// TIA Portal project "CONTROL_ENERGIA" (V12)

(* hardware
DEVICE "S7-300 station_2"  S7-300 station
   slot 0: "Perfil soporte_0"  Rail  6ES7 390-1***0-0AA0
   slot 1: "PS 307 5A_1"  PS 307 5A  6ES7 307-1EA00-0AA0
   slot 2: "CONTROL_ENERGIA"  CPU 314C-2 PN/DP  6ES7 314-6EH04-0AB0  V3.3
      slot 2: "Interfaz PROFINET_1"  PN-IO
         slot 1: "Port_1"  Port
         slot 2: "Port_2"  Port
      slot 5: "DI24/DO16_1"  DI24/DO16
      slot 6: "AI5/AO2_1"  AI5/AO2
      slot 7: "Contaje_1"  Counter
      slot 8: "Posicionamiento_1"  Positioning
   slot 4: "DI8/DO8 x 24V DC / 0,5A_1"  DI8/DO8xDC24V/0.5A  6ES7 323-1BH01-0AA0
*)

// ===== PLC "CONTROL_ENERGIA"  CPU 314C-2 PN/DP =====

VAR_GLOBAL   // PLC tag table "Tabla de variables estándar"
   "Tag_1" AT %I136.0 : Bool;
   "Tag_2" AT %Q136.0 : Bool;
   "Tag_3" AT %I137.0 : Bool;
   "Tag_4" AT %Q136.1 : Bool;
   "Tag_5" AT %I138.0 : Bool;
   "Tag_6" AT %Q137.2 : Bool;
   "Tag_7" AT %Q136.2 : Bool;
   "Tag_8" AT %Q137.0 : Bool;
   "shunt_corriente" AT %IW800 : Int;
   "Tag_10" AT %MW10 : Word;
   "intensidad_medida" AT %MD12 : Real;
   "siempre_cero" AT %M254.0 : Bool;
   "Tag_13" AT %QW800 : Int;
   "Tag_14" AT %MD55 : DWord;
   "consigna salida" AT %MW60 : Int;
   "error_2" AT %MW62 : Word;
   "siempre_uno" AT %M254.1 : Bool;
   "x" AT %MD10 : Real;
   "y" AT %MD20 : Real;
   "x_ala_y" AT %MD30 : Real;
   "intensidad" AT %MD40 : Real;
   "horas" AT %MD50 : Real;
   "intensidad_compensada_peukert" AT %MD60 : Real;
   "rendimiento" AT %MD70 : Real;
   "recarga" AT %MD80 : Real;
   "ret_val_unscale" AT %MW100 : Word;
   "SOC" AT %MD90 : Real;
END_VAR

DATA_BLOCK "parametros_configuracion"   // DB1
{ S7_Optimized_Access := 'FALSE' }
VERSION : 0.1
   VAR
      marca_encendido : Bool;
      Capacidad_fabricante : Real := 625.0;
      Tasa_segun_fabricante : Real := 10.0;
      coeficiente_peukert : Real := 1.13;
      rendimiento_carga : Real := 90.0;
   END_VAR
BEGIN
END_DATA_BLOCK

DATA_BLOCK "Calculo_capacidad_peukert_DB"   // DB2
{ S7_Optimized_Access := 'FALSE' }
VERSION : 0.1
// stored: InstanceOfName Calculo_capacidad_peukert
"Calculo_capacidad_peukert"
BEGIN
END_DATA_BLOCK

DATA_BLOCK "x_a_la_y_DB_intensidad"   // DB3
{ S7_Optimized_Access := 'FALSE' }
VERSION : 0.1
// stored: InstanceOfName x_a_la_y
"x_a_la_y"
BEGIN
END_DATA_BLOCK

DATA_BLOCK "x_a_la_y_DB_capacidad"   // DB4
{ S7_Optimized_Access := 'FALSE' }
VERSION : 0.1
// stored: InstanceOfName x_a_la_y
"x_a_la_y"
BEGIN
END_DATA_BLOCK

DATA_BLOCK "Intensidad_compensada_peukert_DB"   // DB5
{ S7_Optimized_Access := 'FALSE' }
VERSION : 0.1
// stored: InstanceOfName Intensidad_consumida_compensada_peukert
"Intensidad_consumida_compensada_peukert"
BEGIN
END_DATA_BLOCK

DATA_BLOCK "Intensidad_recargada_DB"   // DB6
{ S7_Optimized_Access := 'FALSE' }
VERSION : 0.1
// stored: InstanceOfName Intensidad_recargada
"Intensidad_recargada"
BEGIN
END_DATA_BLOCK

DATA_BLOCK "balance_energetico_DB"   // DB7
{ S7_Optimized_Access := 'FALSE' }
VERSION : 0.1
// stored: InstanceOfName balance_energetico
"balance_energetico"
BEGIN
END_DATA_BLOCK

DATA_BLOCK "S.O.C_DB"   // DB8
{ S7_Optimized_Access := 'FALSE' }
VERSION : 0.1
// stored: InstanceOfName S.O.C
"S.O.C"
BEGIN
END_DATA_BLOCK

FUNCTION_BLOCK "Calculo_capacidad_peukert"   // FB1, LAD
TITLE = calcula por fases la capacidad estandarizada segun peukert Cp=R(C/R)^n
{ S7_Optimized_Access := 'FALSE' }
VERSION : 0.1
   VAR_INPUT
      C : Real;
      R : Real;
      n : Real;
   END_VAR
   VAR_OUTPUT
      CP : Real;
   END_VAR
   VAR_IN_OUT
      "cociente_C/R" : Real;
      parentesis : Real;
   END_VAR
BEGIN

REGION Network 1: Calcula el cociente C/R
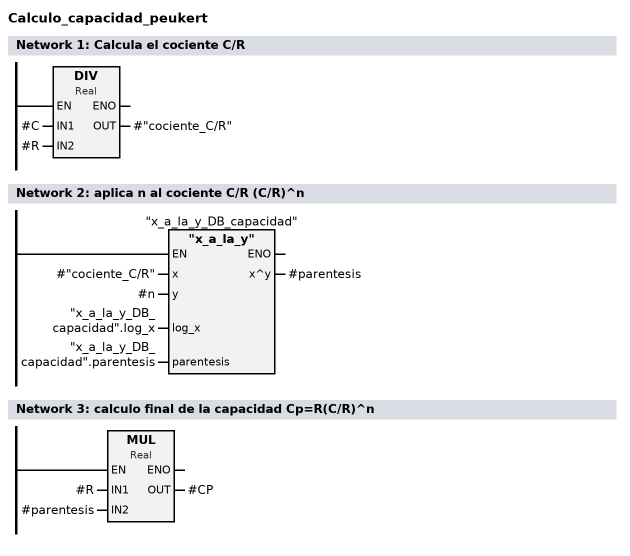
   RUNG wire#powerrail
      { S7_Templates := "SrcType := Real"; S7_GenerateENO := "TRUE" } Div(in1 := #C, in2 := #R, out => #"cociente_C/R")
   END_RUNG
   // the same network as SCL:
   #"cociente_C/R" := #C / #R;
END_REGION

REGION Network 2: aplica n al cociente C/R (C/R)^n
   RUNG wire#powerrail
      "x_a_la_y_DB_capacidad"(x := #"cociente_C/R", y := #n, log_x := "x_a_la_y_DB_capacidad".log_x, parentesis := "x_a_la_y_DB_capacidad".parentesis, "x^y" => #parentesis)
   END_RUNG
   // the same network as SCL:
   "x_a_la_y_DB_capacidad"(x := #"cociente_C/R",   // "x_a_la_y"
                           y := #n,
                           log_x := "x_a_la_y_DB_capacidad".log_x,
                           parentesis := "x_a_la_y_DB_capacidad".parentesis,
                           "x^y" => #parentesis);
END_REGION

REGION Network 3: calculo final de la capacidad Cp=R(C/R)^n
   RUNG wire#powerrail
      { S7_Templates := "SrcType := Real"; S7_GenerateENO := "TRUE" } Mul(in1 := #R, in2 := #parentesis, out => #CP)
   END_RUNG
   // the same network as SCL:
   #CP := #R * #parentesis;
END_REGION
END_FUNCTION_BLOCK

FUNCTION_BLOCK "lectura_intensidad_real"   // FB2, LAD
TITLE = lectura de la intensidad sin compensar
{ S7_Optimized_Access := 'FALSE' }
VERSION : 0.1
BEGIN

REGION Network 1: lectura de la intensidad
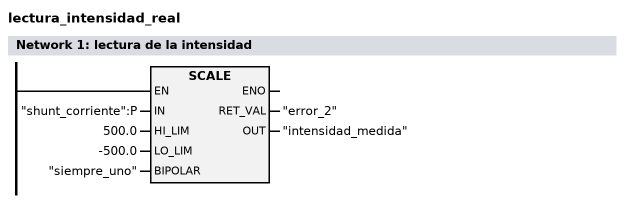
   "error_2" := SCALE(IN := "shunt_corriente":P,
                      HI_LIM := 500.0,
                      LO_LIM := -500.0,
                      BIPOLAR := "siempre_uno",
                      OUT => "intensidad_medida");
END_REGION
END_FUNCTION_BLOCK

FUNCTION_BLOCK "x_a_la_y"   // FB3, LAD
TITLE = calcular trampeando X^Y=EXP(Y*LOG(X))
{ S7_Optimized_Access := 'FALSE' }
VERSION : 0.1
   VAR_INPUT
      x : Real;
      y : Real;
   END_VAR
   VAR_OUTPUT
      "x^y" : Real;
   END_VAR
   VAR_IN_OUT
      log_x : Real;
      parentesis : Real;
   END_VAR
BEGIN

REGION Network 1: LOG(X)
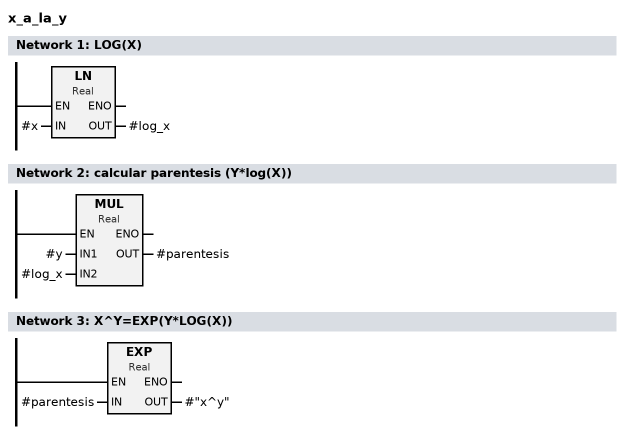
   #log_x := LN(#x);
END_REGION

REGION Network 2: calcular parentesis (Y*log(X))
   RUNG wire#powerrail
      { S7_Templates := "SrcType := Real"; S7_GenerateENO := "TRUE" } Mul(in1 := #y, in2 := #log_x, out => #parentesis)
   END_RUNG
   // the same network as SCL:
   #parentesis := #y * #log_x;
END_REGION

REGION Network 3: X^Y=EXP(Y*LOG(X))
   #"x^y" := EXP(#parentesis);
END_REGION
END_FUNCTION_BLOCK

FUNCTION_BLOCK "Intensidad_consumida_compensada_peukert"   // FB4, LAD
TITLE = Capacidad consumida compensada por Peukert Cp=T*I^n
{ S7_Optimized_Access := 'FALSE' }
VERSION : 0.1
   VAR_INPUT
      tiempo_consumo_horas : Real;
      n : Real;
      intensidad_consumida_amperios : Real;
   END_VAR
   VAR_OUTPUT
      intensidad_compensada : Real;
   END_VAR
   VAR_IN_OUT
      potencia : Real;
      intensidad_absoluta : Real;
   END_VAR
BEGIN

REGION Network 1: sacar el valor absoluto de la I Valores negativos conducen a error
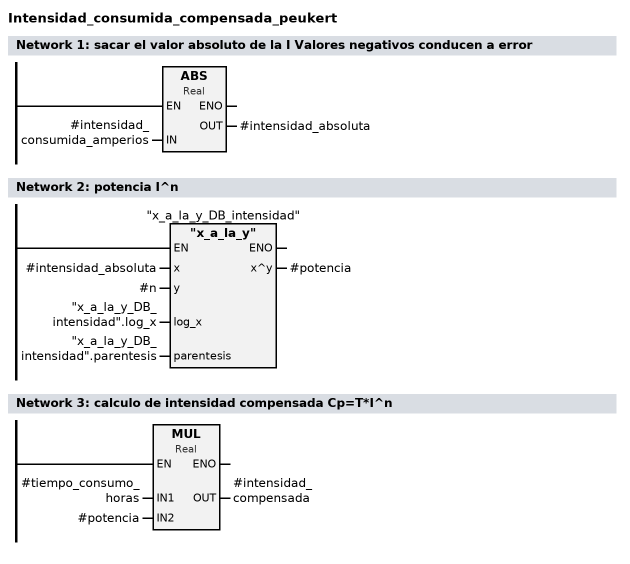
   RUNG wire#powerrail
      { S7_Templates := "SrcType := Real"; S7_GenerateENO := "TRUE" } Abs(in := #intensidad_consumida_amperios, out => #intensidad_absoluta)
   END_RUNG
   // the same network as SCL:
   #intensidad_absoluta := ABS(#intensidad_consumida_amperios);
END_REGION

REGION Network 2: potencia I^n
   RUNG wire#powerrail
      "x_a_la_y_DB_intensidad"(x := #intensidad_absoluta, y := #n, log_x := "x_a_la_y_DB_intensidad".log_x, parentesis := "x_a_la_y_DB_intensidad".parentesis, "x^y" => #potencia)
   END_RUNG
   // the same network as SCL:
   "x_a_la_y_DB_intensidad"(x := #intensidad_absoluta,   // "x_a_la_y"
                           y := #n,
                           log_x := "x_a_la_y_DB_intensidad".log_x,
                           parentesis := "x_a_la_y_DB_intensidad".parentesis,
                           "x^y" => #potencia);
END_REGION

REGION Network 3: calculo de intensidad compensada Cp=T*I^n
   RUNG wire#powerrail
      { S7_Templates := "SrcType := Real"; S7_GenerateENO := "TRUE" } Mul(in1 := #tiempo_consumo_horas, in2 := #potencia, out => #intensidad_compensada)
   END_RUNG
   // the same network as SCL:
   #intensidad_compensada := #tiempo_consumo_horas * #potencia;
END_REGION
END_FUNCTION_BLOCK

FUNCTION_BLOCK "Intensidad_recargada"   // FB5, LAD
TITLE = intensidad entrante aplicado el rendimiento recarga = I*0,X%*tiempo_transcurrido
{ S7_Optimized_Access := 'FALSE' }
VERSION : 0.1
   VAR_INPUT
      intensidad : Real;
      rendimiento : Real;
      tiempo : Real;
   END_VAR
   VAR_IN_OUT
      recarga : Real;
   END_VAR
BEGIN

REGION Network 1: aplica a la recarga el rendimiento configurado
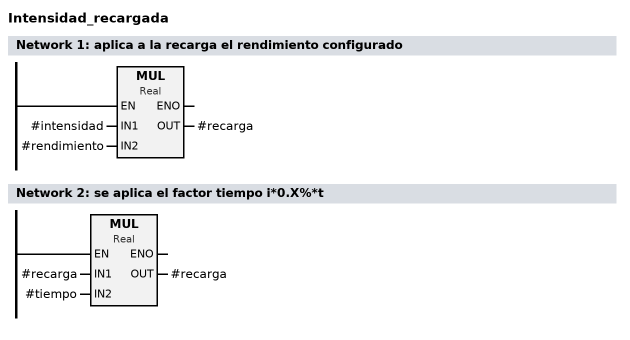
   RUNG wire#powerrail
      { S7_Templates := "SrcType := Real"; S7_GenerateENO := "TRUE" } Mul(in1 := #intensidad, in2 := #rendimiento, out => #recarga)
   END_RUNG
   // the same network as SCL:
   #recarga := #intensidad * #rendimiento;
END_REGION

REGION Network 2: se aplica el factor tiempo i*0.X%*t
   RUNG wire#powerrail
      { S7_Templates := "SrcType := Real"; S7_GenerateENO := "TRUE" } Mul(in1 := #recarga, in2 := #tiempo, out => #recarga)
   END_RUNG
   // the same network as SCL:
   #recarga := #recarga * #tiempo;
END_REGION
END_FUNCTION_BLOCK

FUNCTION_BLOCK "balance_energetico"   // FB6, LAD
TITLE = calcula el balance energetico segun peukert y rendimiento ajustados en parametros
{ S7_Optimized_Access := 'FALSE' }
VERSION : 0.1
   VAR_INPUT
      intensidad_real : Real;
      intensidad_peukert : Real;
      intensidad_carga_comp : Real;
   END_VAR
   VAR_IN_OUT
      intensidad_acumulada : Real;
   END_VAR
BEGIN

REGION Network 1: incrementa la Int acumulada con la int cargada compensada con el rendimiento
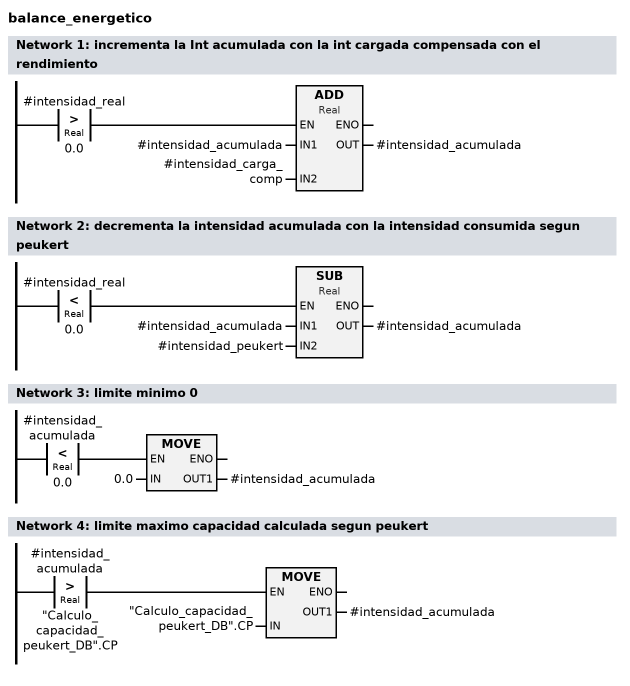
   RUNG wire#powerrail
      { S7_Templates := "SrcType := Real" } GT_Contact(in1 := #intensidad_real, in2 := 0.0)
      { S7_Templates := "SrcType := Real"; S7_GenerateENO := "TRUE" } Add(in1 := #intensidad_acumulada, in2 := #intensidad_carga_comp, out => #intensidad_acumulada)
   END_RUNG
   // the same network as SCL:
   IF #intensidad_real > 0.0 THEN
       #intensidad_acumulada := #intensidad_acumulada + #intensidad_carga_comp;
   END_IF;
END_REGION

REGION Network 2: decrementa la intensidad acumulada con la intensidad consumida segun peukert
   RUNG wire#powerrail
      { S7_Templates := "SrcType := Real" } LT_Contact(in1 := #intensidad_real, in2 := 0.0)
      { S7_Templates := "SrcType := Real"; S7_GenerateENO := "TRUE" } Sub(in1 := #intensidad_acumulada, in2 := #intensidad_peukert, out => #intensidad_acumulada)
   END_RUNG
   // the same network as SCL:
   IF #intensidad_real < 0.0 THEN
       #intensidad_acumulada := #intensidad_acumulada - #intensidad_peukert;
   END_IF;
END_REGION

REGION Network 3: limite minimo 0
   RUNG wire#powerrail
      { S7_Templates := "SrcType := Real" } LT_Contact(in1 := #intensidad_acumulada, in2 := 0.0)
      { S7_GenerateENO := "TRUE" } Move(in := 0.0, out1 => #intensidad_acumulada)
   END_RUNG
   // the same network as SCL:
   IF #intensidad_acumulada < 0.0 THEN #intensidad_acumulada := 0.0; END_IF;
END_REGION

REGION Network 4: limite maximo capacidad calculada segun peukert
   RUNG wire#powerrail
      { S7_Templates := "SrcType := Real" } GT_Contact(in1 := #intensidad_acumulada, in2 := "Calculo_capacidad_peukert_DB".CP)
      { S7_GenerateENO := "TRUE" } Move(in := "Calculo_capacidad_peukert_DB".CP, out1 => #intensidad_acumulada)
   END_RUNG
   // the same network as SCL:
   IF #intensidad_acumulada > "Calculo_capacidad_peukert_DB".CP THEN
       #intensidad_acumulada := "Calculo_capacidad_peukert_DB".CP;
   END_IF;
END_REGION
END_FUNCTION_BLOCK

FUNCTION_BLOCK "S.O.C"   // FB7, LAD
{ S7_Optimized_Access := 'FALSE' }
VERSION : 0.1
   VAR_INPUT
      "intensidad_acumulada." : Real;
   END_VAR
   VAR_OUTPUT
      SOC : Real;
   END_VAR
   VAR_IN_OUT
      intensidad_integer : Int;
   END_VAR
BEGIN

REGION Network 1: convertimos la intensidad de real a entero
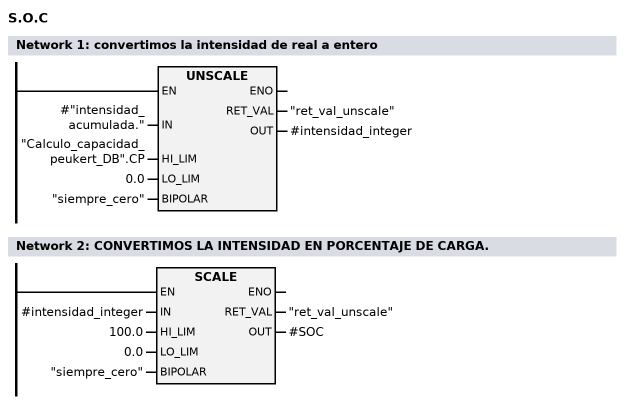
   "ret_val_unscale" := UNSCALE(IN := #"intensidad_acumulada.",
                           HI_LIM := "Calculo_capacidad_peukert_DB".CP,
                           LO_LIM := 0.0,
                           BIPOLAR := "siempre_cero",
                           OUT => #intensidad_integer);
END_REGION

REGION Network 2: CONVERTIMOS LA INTENSIDAD EN PORCENTAJE DE CARGA.
   "ret_val_unscale" := SCALE(IN := #intensidad_integer,
                           HI_LIM := 100.0,
                           LO_LIM := 0.0,
                           BIPOLAR := "siempre_cero",
                           OUT => #SOC);
END_REGION
END_FUNCTION_BLOCK

ORGANIZATION_BLOCK "Main"   // OB1, LAD
TITLE = "Main Program Sweep (Cycle)"
{ S7_Optimized_Access := 'FALSE' }
VERSION : 0.1
   VAR_TEMP
      OB1_EV_CLASS : Byte;   // Bits 0-3 = 1 (Coming event), Bits 4-7 = 1 (Event class 1)
      OB1_SCAN_1 : Byte;   // 1 (Cold restart scan 1 of OB 1), 3 (Scan 2-n of OB 1)
      OB1_PRIORITY : Byte;   // Priority of OB Execution
      OB1_OB_NUMBR : Byte;   // 1 (Organization block 1, OB1)
      OB1_RESERVED_1 : Byte;   // Reserved for system
      OB1_RESERVED_2 : Byte;   // Reserved for system
      OB1_PREV_CYCLE : Int;   // Cycle time of previous OB1 scan (milliseconds)
      OB1_MIN_CYCLE : Int;   // Minimum cycle time of OB1 (milliseconds)
      OB1_MAX_CYCLE : Int;   // Maximum cycle time of OB1 (milliseconds)
      OB1_DATE_TIME : Date_And_Time;   // Date and time OB1 started
   END_VAR
BEGIN

REGION Network 1: prueba calculo capacidad peukert
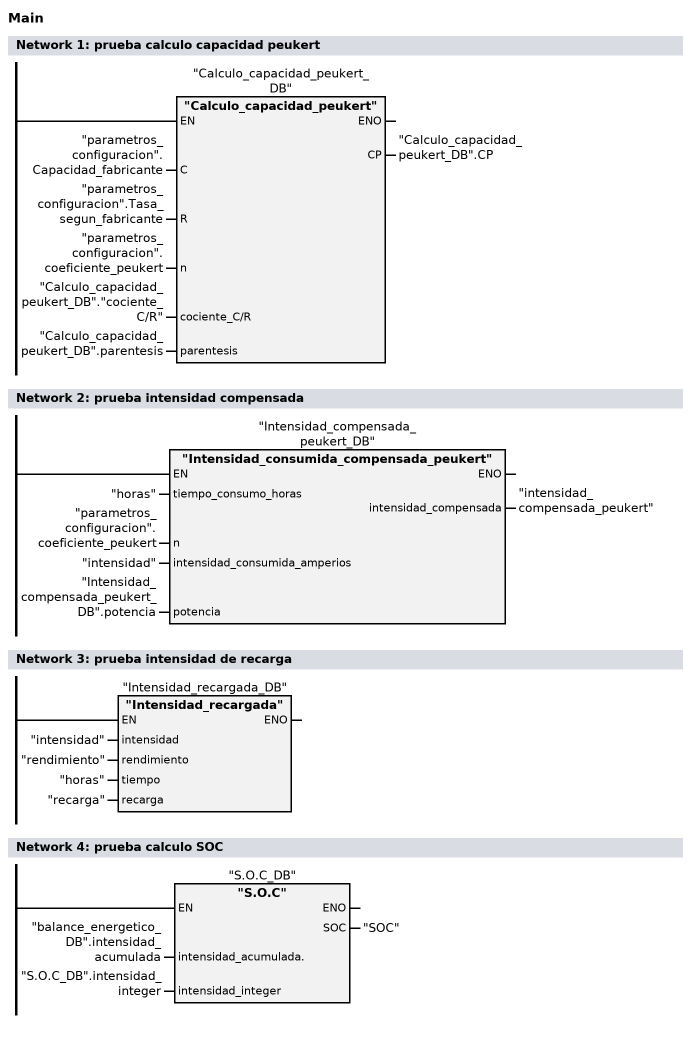
   RUNG wire#powerrail
      "Calculo_capacidad_peukert_DB"(C := "parametros_configuracion".Capacidad_fabricante, R := "parametros_configuracion".Tasa_segun_fabricante, n := "parametros_configuracion".coeficiente_peukert, "cociente_C/R" := "Calculo_capacidad_peukert_DB"."cociente_C/R", parentesis := "Calculo_capacidad_peukert_DB".parentesis, CP => "Calculo_capacidad_peukert_DB".CP)
   END_RUNG
   // the same network as SCL:
   "Calculo_capacidad_peukert_DB"(C := "parametros_configuracion".Capacidad_fabricante,   // "Calculo_capacidad_peukert"
                           R := "parametros_configuracion".Tasa_segun_fabricante,
                           n := "parametros_configuracion".coeficiente_peukert,
                           "cociente_C/R" := "Calculo_capacidad_peukert_DB"."cociente_C/R",
                           parentesis := "Calculo_capacidad_peukert_DB".parentesis,
                           CP => "Calculo_capacidad_peukert_DB".CP);
END_REGION

REGION Network 2: prueba intensidad compensada
   RUNG wire#powerrail
      "Intensidad_compensada_peukert_DB"(tiempo_consumo_horas := "horas", n := "parametros_configuracion".coeficiente_peukert, potencia := "Intensidad_compensada_peukert_DB".potencia, intensidad_consumida_amperios := "intensidad", intensidad_compensada => "intensidad_compensada_peukert")
   END_RUNG
   // the same network as SCL:
   "Intensidad_compensada_peukert_DB"(tiempo_consumo_horas := "horas",   // "Intensidad_consumida_compensada_peukert"
                           n := "parametros_configuracion".coeficiente_peukert,
                           intensidad_consumida_amperios := "intensidad",
                           potencia := "Intensidad_compensada_peukert_DB".potencia,
                           intensidad_compensada => "intensidad_compensada_peukert");
END_REGION

REGION Network 3: prueba intensidad de recarga
   RUNG wire#powerrail
      "Intensidad_recargada_DB"(intensidad := "intensidad", rendimiento := "rendimiento", tiempo := "horas", recarga := "recarga")
   END_RUNG
   // the same network as SCL:
   "Intensidad_recargada_DB"(intensidad := "intensidad",   // "Intensidad_recargada"
                           rendimiento := "rendimiento",
                           tiempo := "horas",
                           recarga := "recarga");
END_REGION

REGION Network 4: prueba calculo SOC
   RUNG wire#powerrail
      "S.O.C_DB"("intensidad_acumulada." := "balance_energetico_DB".intensidad_acumulada, intensidad_integer := "S.O.C_DB".intensidad_integer, SOC => "SOC")
   END_RUNG
   // the same network as SCL:
   "S.O.C_DB"("intensidad_acumulada." := "balance_energetico_DB".intensidad_acumulada,   // "S.O.C"
              intensidad_integer := "S.O.C_DB".intensidad_integer,
              SOC => "SOC");
END_REGION
END_ORGANIZATION_BLOCK

ORGANIZATION_BLOCK "SAMPLER"   // OB32, LAD
TITLE = "Cyclic Interrupt"
{ S7_Optimized_Access := 'FALSE' }
VERSION : 0.1
   VAR_TEMP
      OB32_EV_CLASS : Byte;   // Bits 0-3 = 1 (Coming event), Bits 4-7 = 1 (Event class 1)
      OB32_STRT_INF : Byte;   // 16#33 (OB 32 has started)
      OB32_PRIORITY : Byte;   // Priority of OB Execution
      OB32_OB_NUMBR : Byte;   // 32 (Organization block 32, OB32)
      OB32_RESERVED_1 : Byte;   // Reserved for system
      OB32_RESERVED_2 : Byte;   // Reserved for system
      OB32_PHS_OFFSET : Int;   // Phase offset (integer, milliseconds)
      OB32_RESERVED_3 : Int;   // Reserved for system
      OB32_EXC_FREQ : Int;   // Frequency of execution (msec)
      OB32_DATE_TIME : Date_And_Time;   // Date and time OB32 started
   END_VAR
BEGIN

REGION Network 1: calcula balance energetico usando las I calculadas y el factor tiempo (tiempo sampler)
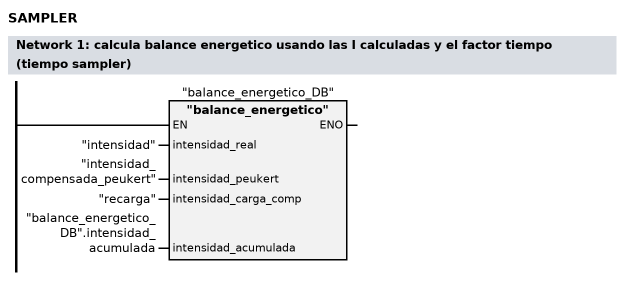
   RUNG wire#powerrail
      "balance_energetico_DB"(intensidad_real := "intensidad", intensidad_peukert := "intensidad_compensada_peukert", intensidad_carga_comp := "recarga", intensidad_acumulada := "balance_energetico_DB".intensidad_acumulada)
   END_RUNG
   // the same network as SCL:
   "balance_energetico_DB"(intensidad_real := "intensidad",   // "balance_energetico"
                           intensidad_peukert := "intensidad_compensada_peukert",
                           intensidad_carga_comp := "recarga",
                           intensidad_acumulada := "balance_energetico_DB".intensidad_acumulada);
END_REGION
END_ORGANIZATION_BLOCK

ORGANIZATION_BLOCK "CYCL_FLT"   // OB80, LAD
TITLE = "Cycle Time Fault"
{ S7_Optimized_Access := 'FALSE' }
VERSION : 0.1
   VAR_TEMP
      OB80_EV_CLASS : Byte;   // 16#35, Event class 3, Entering event state, Internal fault event
      OB80_FLT_ID : Byte;   // 16#XX, Fault identifcation code
      OB80_PRIORITY : Byte;   // Priority of OB Execution
      OB80_OB_NUMBR : Byte;   // 80 (Organization block 80, OB80)
      OB80_RESERVED_1 : Byte;   // Reserved for system
      OB80_RESERVED_2 : Byte;   // Reserved for system
      OB80_ERROR_INFO : Word;   // Error information on event
      OB80_ERR_EV_CLASS : Byte;   // Class of event causing error
      OB80_ERR_EV_NUM : Byte;   // Number of event causing error
      OB80_OB_PRIORITY : Byte;   // Priority of OB causing error
      OB80_OB_NUM : Byte;   // Number of OB causing error
      OB80_DATE_TIME : Date_And_Time;   // Date and time OB80 started
   END_VAR
BEGIN
END_ORGANIZATION_BLOCK

ORGANIZATION_BLOCK "I/O_FLT1"   // OB82, LAD
TITLE = "I/O Point Fault"
{ S7_Optimized_Access := 'FALSE' }
VERSION : 0.1
   VAR_TEMP
      OB82_EV_CLASS : Byte;   // 16#39, Event class 3, Entering event state, Internal fault event
      OB82_FLT_ID : Byte;   // 16#XX, Fault identifcation code
      OB82_PRIORITY : Byte;   // Priority of OB Execution
      OB82_OB_NUMBR : Byte;   // 82 (Organization block 82, OB82)
      OB82_RESERVED_1 : Byte;   // Reserved for system
      OB82_IO_FLAG : Byte;   // Input (01010100), Output (01010101)
      OB82_MDL_ADDR : Word;   // Base address of module with fault
      OB82_MDL_DEFECT : Bool;   // Module defective
      OB82_INT_FAULT : Bool;   // Internal fault
      OB82_EXT_FAULT : Bool;   // External fault
      OB82_PNT_INFO : Bool;   // Point information
      OB82_EXT_VOLTAGE : Bool;   // External voltage low
      OB82_FLD_CONNCTR : Bool;   // Field wiring connector missing
      OB82_NO_CONFIG : Bool;   // Module has no configuration data
      OB82_CONFIG_ERR : Bool;   // Module has configuration error
      OB82_MDL_TYPE : Byte;   // Type of module
      OB82_SUB_MDL_ERR : Bool;   // Sub-Module is missing or has error
      OB82_COMM_FAULT : Bool;   // Communication fault
      OB82_MDL_STOP : Bool;   // Module is stopped
      OB82_WTCH_DOG_FLT : Bool;   // Watch dog timer stopped module
      OB82_INT_PS_FLT : Bool;   // Internal power supply fault
      OB82_PRIM_BATT_FLT : Bool;   // Primary battery is in fault
      OB82_BCKUP_BATT_FLT : Bool;   // Backup battery is in fault
      OB82_RESERVED_2 : Bool;   // Reserved for system
      OB82_RACK_FLT : Bool;   // Rack fault, only for bus interface module
      OB82_PROC_FLT : Bool;   // Processor fault
      OB82_EPROM_FLT : Bool;   // EPROM fault
      OB82_RAM_FLT : Bool;   // RAM fault
      OB82_ADU_FLT : Bool;   // ADU fault
      OB82_FUSE_FLT : Bool;   // Fuse fault
      OB82_HW_INTR_FLT : Bool;   // Hardware interupt input in fault
      OB82_RESERVED_3 : Bool;   // Reserved for system
      OB82_DATE_TIME : Date_And_Time;   // Date and time OB82 started
   END_VAR
BEGIN
END_ORGANIZATION_BLOCK

ORGANIZATION_BLOCK "I/O_FLT2"   // OB83, LAD
TITLE = "I/O Point Fault"
{ S7_Optimized_Access := 'FALSE' }
VERSION : 0.1
   VAR_TEMP
      OB83_EV_CLASS : Byte;   // 16#38/39, Event class 3, module inserted/removed (8/9)
      OB83_FLT_ID : Byte;   // 16#XX, Fault identifcation code
      OB83_PRIORITY : Byte;   // Priority of OB Execution
      OB83_OB_NUMBR : Byte;   // 83 (Organization block 83, OB83)
      OB83_RESERVED_1 : Byte;   // Reserved for system
      OB83_MDL_ID : Byte;   // Input module (01010100), Output module (01010101)
      OB83_MDL_ADDR : Word;   // Base address of module with point fault
      OB83_RACK_NUM : Int;   // Number of rack that has module with point fault
      OB83_MDL_TYPE : Word;   // Module type with point fault
      OB83_DATE_TIME : Date_And_Time;   // Date and time OB83 started
   END_VAR
BEGIN
END_ORGANIZATION_BLOCK

ORGANIZATION_BLOCK "OBNL_FLT"   // OB85, LAD
TITLE = "Organization Block (OB) Not Loaded Fault"
{ S7_Optimized_Access := 'FALSE' }
VERSION : 0.1
   VAR_TEMP
      OB85_EV_CLASS : Byte;   // 16#35 Event class 3
      OB85_FLT_ID : Byte;   // 16#XX, Fault identification code
      OB85_PRIORITY : Byte;   // Priority of OB Execution
      OB85_OB_NUMBR : Byte;   // 85 (Organization block 85, OB85)
      OB85_RESERVED_1 : Byte;   // Reserved for system
      OB85_RESERVED_2 : Byte;   // Reserved for system
      OB85_RESERVED_3 : Int;   // Reserved for system
      OB85_ERR_EV_CLASS : Byte;   // Class of event causing error
      OB85_ERR_EV_NUM : Byte;   // Number of event causing error
      OB85_OB_PRIOR : Byte;   // Priority of OB causing error
      OB85_OB_NUM : Byte;   // Number of OB causing error
      OB85_DATE_TIME : Date_And_Time;   // Date and time OB85 started
   END_VAR
BEGIN
END_ORGANIZATION_BLOCK

ORGANIZATION_BLOCK "COMPLETE RESTART"   // OB100, LAD
TITLE = "Complete Restart"
{ S7_Optimized_Access := 'FALSE' }
VERSION : 0.1
   VAR_TEMP
      OB100_EV_CLASS : Byte;   // 16#13, Event class 1, Entering event state, Event logged in diagnostic buffer
      OB100_STRTUP : Byte;   // 16#81/82/83/84 Method of startup
      OB100_PRIORITY : Byte;   // Priority of OB Execution
      OB100_OB_NUMBR : Byte;   // 100 (Organization block 100, OB100)
      OB100_RESERVED_1 : Byte;   // Reserved for system
      OB100_RESERVED_2 : Byte;   // Reserved for system
      OB100_STOP : Word;   // Event that caused CPU to stop (16#4xxx)
      OB100_STRT_INFO : DWord;   // Information on how system started
      OB100_DATE_TIME : Date_And_Time;   // Date and time OB100 started
   END_VAR
BEGIN

REGION Network 1: Crear Cero
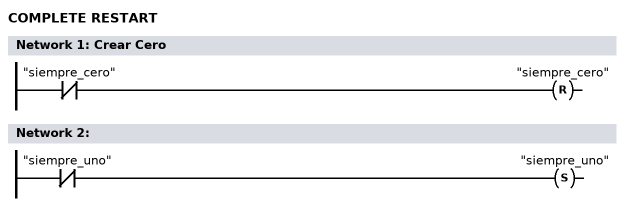
   RUNG wire#powerrail
      I_Contact( "siempre_cero" )
      R_Coil( "siempre_cero" )
   END_RUNG
   // the same network as SCL:
   IF NOT "siempre_cero" THEN "siempre_cero" := FALSE; END_IF;
END_REGION

REGION Network 2
   RUNG wire#powerrail
      I_Contact( "siempre_uno" )
      S_Coil( "siempre_uno" )
   END_RUNG
   // the same network as SCL:
   IF NOT "siempre_uno" THEN "siempre_uno" := TRUE; END_IF;
END_REGION
END_ORGANIZATION_BLOCK

ORGANIZATION_BLOCK "PROG_ERR"   // OB121, LAD
TITLE = "Programming Error"
{ S7_Optimized_Access := 'FALSE' }
VERSION : 0.1
   VAR_TEMP
      OB121_EV_CLASS : Byte;   // 16#25, Event class 2, Entering event state, Internal fault event
      OB121_SW_FLT : Byte;   // 16#XX Software programming fault
      OB121_PRIORITY : Byte;   // Priority of OB Execution
      OB121_OB_NUMBR : Byte;   // 121 (Organization block 121, OB121)
      OB121_BLK_TYPE : Byte;   // 16#88/8A/8B/8C/8E Type of block fault occured in
      OB121_RESERVED_1 : Byte;   // Reserved for system
      OB121_FLT_REG : Word;   // 16#XX Specific register that caused fault
      OB121_BLK_NUM : Word;   // Number of block that programming fault occured in
      OB121_PRG_ADDR : Word;   // Address in block where programming fault occured
      OB121_DATE_TIME : Date_And_Time;   // Date and time OB121 started
   END_VAR
BEGIN
END_ORGANIZATION_BLOCK